(* CODESYS project 03_WagoApp_1.10.0.x_Datalogger_Example_Training_01.project

Project tree, tasks and I/O mapping:
  PFC200_G2_2ETH_RS : 750-8212 PFC200 G2 2ETH RS, WAGO, order no. 0750-8212, version 5.16.3.46
    application Application
      libraries: ; WagoAppDatalogger, 1.0.4.0 (WAGO); Util, * (System); VisuDialogs, * (System)
      task PLC_Task (cyclic, interval 1000 ms, priority 15) calls PLC_PRG
      task VISU_TASK (cyclic, interval 100 ms, priority 15) calls VisuElems.Visu_Prg
      program PLC_PRG [FBD]: INIT
      visualisation Datalogger
      global variables PersistentVars
    ProjectConfiguration
    Kbus : Kbus, WAGO, version 1.4.0.2
        settings: program start interlock = True
        unmapped channels: K-BUS diagnostics
    MODBUS
      MODBUS : MODBUS, WAGO, order no. n/a, version 1.1.1.16
    Serial
      COM1 : COM1, WAGO, version 0.0.0.19
    Common.PCI
    EtherNet/IP
      Ethernet : Ethernet, WAGO, version 35.16.0.0
          settings: IPAddress = [192, 168, 1, 106]; SubnetMask = [0, 0, 0, 0]; MACAddress = [16#00, 16#00, 16#00, 16#00, 16#00, 16#00]; NetworkInterfaceName = 'br0'; NetworkInterfaceName = "br0"
  libraries: VisuSymbols, 3.5.17.0 (System); WagoVisuIcons, 1.1.0.4 (WAGO)
  text list GlobalTextList
  00000000-0000-0000-0000-000000000000|C:\Users\u0100068\AppData\Local\Temp\110df24e080145dea3de34d6366c2e37\e868b832187f4f1a859da50215710801\Project.xml
*)

// PFC200_G2_2ETH_RS/Application/PersistentVars
{attribute 'qualified_only'}
VAR_GLOBAL PERSISTENT RETAIN
	// Instanzpfad der persistenten Variablen erzeugt
	PLC_PRG.aChannels: ARRAY [1..WagoAppDatalogger.MAX_CHANNELS] OF REAL;
	// Instanzpfad der persistenten Variablen erzeugt
	PLC_PRG.typConfigParameters: WagoAppDatalogger.typConfigDatalogger;
	// Instanzpfad der persistenten Variablen erzeugt
	PLC_PRG.tCosinePeriod: TIME := TIME#30s0ms;
	// Instanzpfad der persistenten Variablen erzeugt
	PLC_PRG.tSinusPeriod: TIME := TIME#1m0s0ms;
END_VAR

// PFC200_G2_2ETH_RS/Application/PLC_PRG
PROGRAM PLC_PRG
VAR
	_oFbDatalogger			: WagoAppDatalogger.FbDatalogger;
		xEnable				: BOOL:=TRUE;
		xEvent				: BOOL;
		sStatusDatalogger	: STRING;
		xReady				: BOOL;
	Generator1				: Util.GEN;
		xReset	  			: BOOL;
		SINUS				: Util.GEN_MODE := 5;
	Generator2				: Util.GEN;
		COSINUS				: Util.GEN_MODE := 6;
	//Variables for INIT
		xFirstCycle			: BOOL := TRUE;
		i					: INT;
	
	iSinusAmplitude: INT := 400;
	iCosinusAmplitude: INT := 400;
END_VAR
VAR RETAIN PERSISTENT
		aChannels 			: ARRAY [1..WagoAppDatalogger.MAX_CHANNELS] OF REAL;
		typConfigParameters	: WagoAppDatalogger.typConfigDatalogger;
		tCosinePeriod: TIME := T#30S;
		tSinusPeriod: TIME := T#60S;
END_VAR

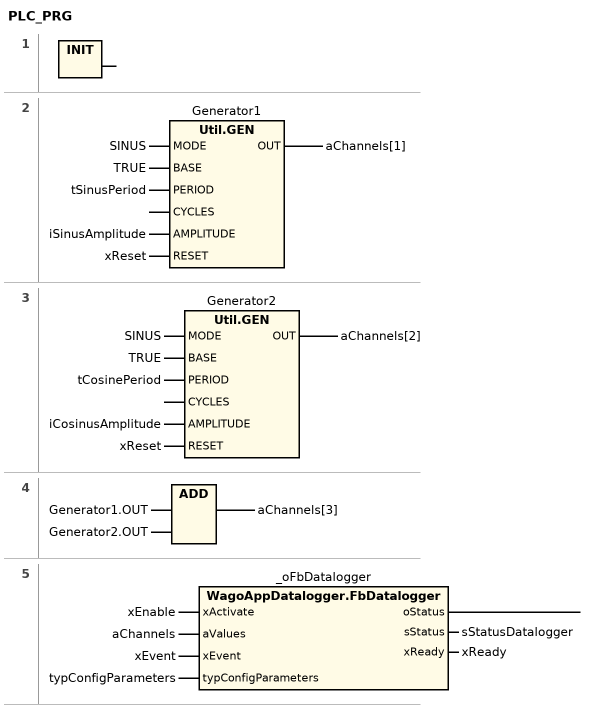
// NETWORK 1
INIT();

// NETWORK 2
Generator1(
    MODE := SINUS,
    BASE := TRUE,
    PERIOD := tSinusPeriod,
    AMPLITUDE := iSinusAmplitude,
    RESET := xReset); // Util.GEN
aChannels[1] := Generator1.OUT;

// NETWORK 3
Generator2(
    MODE := SINUS,
    BASE := TRUE,
    PERIOD := tCosinePeriod,
    AMPLITUDE := iCosinusAmplitude,
    RESET := xReset); // Util.GEN
aChannels[2] := Generator2.OUT;

// NETWORK 4
aChannels[3] := Generator1.OUT + Generator2.OUT;

// NETWORK 5
_oFbDatalogger(
    xActivate := xEnable,
    aValues := aChannels,
    xEvent := xEvent,
    typConfigParameters := typConfigParameters,
    sStatus => sStatusDatalogger,
    xReady => xReady); // WagoAppDatalogger.FbDatalogger

ACTION INIT:
IF xFirstCycle THEN
	typConfigParameters.bInterval				:= 3;
	typConfigParameters.uiIntervalFactor		:= 1;
	typConfigParameters.sFilename				:= 'Logfile.csv';
	typConfigParameters.sPath					:= '/media/sd/CSV_Files/';
	typConfigParameters.xAppendDate				:= TRUE;
	typConfigParameters.xCyclicLogging			:= TRUE;
	typConfigParameters.sDecimalSeparator		:= ',';
	typConfigParameters.sColumnSeparator		:= ';';

//Will be executed only once after start of program to enable editable channel variables 
	//Set all Channels to false
	FOR i:=1 TO 80 DO
		typConfigParameters.atypChannelConfig[i].xChannelExists	:= FALSE;
	END_FOR

	typConfigParameters.atypChannelConfig[1].xChannelExists		:= TRUE;
	typConfigParameters.atypChannelConfig[1].sChannelName		:= '1st Sinus Curve';
	typConfigParameters.atypChannelConfig[1].sUnit				:= 'V';
	typConfigParameters.atypChannelConfig[1].bDecimalPlaces		:= 2;			//number of digits afer decimal-point. IF not specified: Default-Value = 2
	typConfigParameters.atypChannelConfig[1].xLogAlarm			:= TRUE;		//Shows alarm column of sine-function in file (for Standard-Datalogger) 
	typConfigParameters.atypChannelConfig[1].rAlarmLowerLimit	:= -380;
	typConfigParameters.atypChannelConfig[1].rAlarmUpperLimit	:= 380;

	typConfigParameters.atypChannelConfig[2].xChannelExists		:= TRUE;
	typConfigParameters.atypChannelConfig[2].sChannelName		:= '2nd Sinus Curve';
	typConfigParameters.atypChannelConfig[2].sUnit				:= 'V';
	typConfigParameters.atypChannelConfig[2].bDecimalPlaces		:= 2;			//number of digits afer decimal-point. IF not specified: Default-Value = 2
	typConfigParameters.atypChannelConfig[2].xLogAlarm			:= TRUE;		//Shows alarm column of sine-function in file (for Standard-Datalogger) 
	typConfigParameters.atypChannelConfig[2].rAlarmLowerLimit	:= -380;
	typConfigParameters.atypChannelConfig[2].rAlarmUpperLimit	:= 380;

	typConfigParameters.atypChannelConfig[3].xChannelExists		:= TRUE;
	typConfigParameters.atypChannelConfig[3].sChannelName		:= 'Beat Curve';
	typConfigParameters.atypChannelConfig[3].sUnit				:= 'V';
	typConfigParameters.atypChannelConfig[3].bDecimalPlaces		:= 2;			//number of digits afer decimal-point. IF not specified: Default-Value = 2
	typConfigParameters.atypChannelConfig[3].xLogAlarm			:= TRUE;		//Shows alarm column of sine-function in file (for Standard-Datalogger) 
	typConfigParameters.atypChannelConfig[3].rAlarmLowerLimit	:= -500;
	typConfigParameters.atypChannelConfig[3].rAlarmUpperLimit	:= 500;
	

	xFirstCycle					:= FALSE;										//Prevents another call of initialization 
END_IF

//Entries outside of IF-THEN construct will be executed in each cycle of the PLC
END_ACTION

END_PROGRAM

// PFC200_G2_2ETH_RS/Application/Datalogger
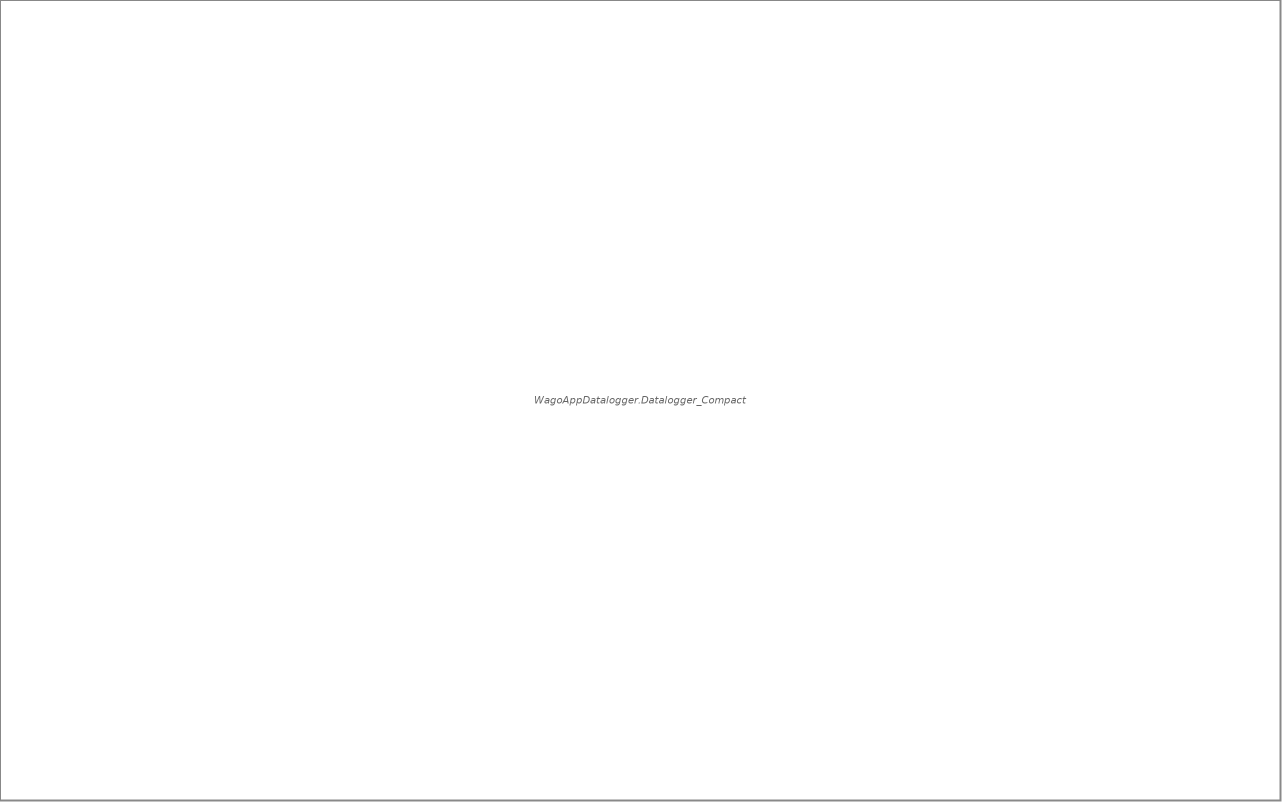
VISUALIZATION Datalogger  // 1282x802
    Frame (0,0 1280x800)
        shows WagoAppDatalogger.Datalogger_Compact(oDatalogger := PLC_PRG._oFbDatalogger)
END_VISUALIZATION
